# EPICS alarm handler configuration: alh_files/mgnt_li30.alhConfig
GROUP NULL MGNT:LI30:1
   $COMMAND edm -x -eolc -noedit mgnt_li30_main.edl

$ALIAS LI30
$GUIDANCE
LI30 Magnets
   Group Name: MGNT:LI30:1
   Summary PV:  MGNT:LI30:1:STATSUMY
$END

   INCLUDE MGNT:LI30:1 ./mgnt_li30_lgps.alhConfig
   INCLUDE MGNT:LI30:1 ./mgnt_li30_quad.alhConfig
   INCLUDE MGNT:LI30:1 ./mgnt_li30_xcor.alhConfig
   INCLUDE MGNT:LI30:1 ./mgnt_li30_ycor.alhConfig
